// NETWORK 2
//   _strobeTimer.ET: elapsed time
Control.SystemTime.FastFlash := F_LIMIT(En := TRUE, High := 500, Value := TIME_TO_REAL(_strobeTimer.ET), Low := 0) OR F_LIMIT(En := TRUE, High := 1500, Value := TIME_TO_REAL(_strobeTimer.ET), Low := 1000);

// NETWORK 3
//   _strobeTimer.ET: elapsed time
Control.SystemTime.PulseFlash := F_LIMIT(En := TRUE, High := 1500, Value := TIME_TO_REAL(_strobeTimer.ET), Low := 1250) OR F_LIMIT(En := TRUE, High := 2000, Value := TIME_TO_REAL(_strobeTimer.ET), Low := 1750);

// NETWORK 4
//   _strobeTimer.ET: elapsed time
Control.SystemTime.SlowFlash := F_LIMIT(En := TRUE, High := 1000, Value := TIME_TO_REAL(_strobeTimer.ET), Low := 0);
END_ACTION

ACTION A_SyncSystemTime:
_fb_LocalSystemTime(sNetID := '', bEnable := TRUE, dwCycle := 15, dwOpt := 1, tTimeout := DEFAULT_ADS_TIMEOUT);
IF _fb_LocalSystemTime.bValid THEN
	Control.SystemTime.CurrentTime := _fb_LocalSystemTime.systemTime;
END_IF
END_ACTION

ACTION A_TimePulses:
//Second Pulse
_timer_ET := _timer_ET + DWORD_TO_DINT(_lastScanTime);
IF _timer_ET >= _ticksInSecond THEN 
	Control.SystemTime.SecondPulse := TRUE;
	Control.SystemTime.SecondsNow := TO_DWORD(SYSTEMTIME_TO_DT(Control.SystemTime.CurrentTime));
	_timer_ET := 0;
ELSE
	Control.SystemTime.SecondPulse := FALSE;
END_IF

//Minute Pulse
_MinutePulse(CLK := Control.SystemTime.CurrentTime.wSecond = 0);
Control.SystemTime.MinutePulse :=  _MinutePulse.Q;

//Hour Pulse
_HourPulse(CLK := Control.SystemTime.CurrentTime.wMinute = 0);
Control.SystemTime.HourPulse :=  _HourPulse.Q;

//Midnight Pulse
IF WORD_TO_INT(Control.SystemTime.CurrentTime.wDay) <> Control_SP.TimeManagement.PreviousDay THEN
	Control.SystemTime.MidnightPulse := TRUE;
	Control_SP.TimeManagement.PreviousDay := WORD_TO_INT(Control.SystemTime.CurrentTime.wDay);
ELSE
	Control.SystemTime.MidnightPulse := FALSE;
END_IF
END_ACTION

ACTION A_UpTime:
IF Control.SystemTime.SecondPulse THEN
	//Up time since last reset
	Control.SystemTime.UpTime.Seconds := Control.SystemTime.UpTime.Seconds + 1;
	IF Control.SystemTime.UpTime.Seconds >= 60 THEN 
		Control.SystemTime.UpTime.Minutes := Control.SystemTime.UpTime.Minutes + 1;
		Control.SystemTime.UpTime.Seconds := 0;
	END_IF
	IF Control.SystemTime.UpTime.Minutes >= 60 THEN 
		Control.SystemTime.UpTime.Hours := Control.SystemTime.UpTime.Hours + 1;
		Control.SystemTime.UpTime.Minutes := 0;
	END_IF
	IF Control.SystemTime.UpTime.Hours >= 24 THEN 
		Control.SystemTime.UpTime.Days := Control.SystemTime.UpTime.Days + 1;
		Control.SystemTime.UpTime.Hours := 0;
	END_IF
	
	//Total up time
	Control_SP.TimeManagement.TotalUpTime.Seconds := Control_SP.TimeManagement.TotalUpTime.Seconds + 1;
	IF Control_SP.TimeManagement.TotalUpTime.Seconds >= 60 THEN 
		Control_SP.TimeManagement.TotalUpTime.Minutes := Control_SP.TimeManagement.TotalUpTime.Minutes + 1;
		Control_SP.TimeManagement.TotalUpTime.Seconds := 0;
	END_IF
	IF Control_SP.TimeManagement.TotalUpTime.Minutes >= 60 THEN 
		Control_SP.TimeManagement.TotalUpTime.Hours := Control_SP.TimeManagement.TotalUpTime.Hours + 1;
		Control_SP.TimeManagement.TotalUpTime.Minutes := 0;
	END_IF
	IF Control_SP.TimeManagement.TotalUpTime.Hours >= 24 THEN 
		Control_SP.TimeManagement.TotalUpTime.Days := Control_SP.TimeManagement.TotalUpTime.Days + 1;
		Control_SP.TimeManagement.TotalUpTime.Hours := 0;
	END_IF
END_IF
END_ACTION

END_FUNCTION_BLOCK

// Objects/FB_TwinSAFE_V4_01/FB_TwinSAFE
FUNCTION_BLOCK FINAL FB_TwinSAFE EXTENDS FB_EventLogger
VAR_IN_OUT
	Control								: ST_System;
END_VAR
VAR
	_ComErr					AT %I*		: BOOL;
	_FbErr					AT %I*		: BOOL;
	_OutErr					AT %I*		: BOOL;
	_ComStartUp				AT %I*		: BOOL;
	_OtherErr				AT %I*		: BOOL;
	_State					AT %I*		: UINT;
	_Daig					AT %I*		: UINT;
	_FSOUTModule1Fault 		AT %I* 		: BOOL;
	_FSOUTModule2Fault 		AT %I* 		: BOOL;
	_FSOUTModule3Fault 		AT %I* 		: BOOL;
	_FSOUTModule4Fault 		AT %I* 		: BOOL;
	_FSOUTModule5Fault 		AT %I* 		: BOOL;
	_FSOUTModule6Fault 		AT %I* 		: BOOL;
	_FSOUTRelaisModuleFault AT %I*      : BOOL;
	_FSINModule1Fault		AT %I* 		: BOOL;
	_FSINModule2Fault		AT %I* 		: BOOL;
	_FSINModule3Fault		AT %I* 		: BOOL;
	_FSINModule4Fault		AT %I* 		: BOOL;
	_FSINModule5Fault		AT %I* 		: BOOL;
	_FSINModule6Fault		AT %I* 		: BOOL;
	_FSINModule7Fault		AT %I* 		: BOOL;
	_FSINModule8Fault		AT %I* 		: BOOL;
	_FSINModule9Fault		AT %I* 		: BOOL;
	_FSINModule10Fault		AT %I* 		: BOOL;
	_SafetyChainFault 	    AT %I*  	: BOOL;
	_SafetyInRun			AT %I*  	: BOOL;
	_Module1Fault			AT %I*  	: BOOL;
	_RunStop				AT %Q*		: BOOL;
	_ErrAck					AT %Q*		: BOOL;
	_SafetyInRunReturn		AT %Q*  	: BOOL;
	_ModuleFault					  	: BOOL;
	_Alarm								: BOOL;					
	_Warning							: BOOL;					
	_AlarmMute							: BOOL;					
	_AlarmNum							: DINT;					
	_WarningNum							: DINT;					
	_FaultTimer_ET						: REAL;	
	_r_Trig								: ARRAY[0..9] OF R_TRIG;
END_VAR
VAR PERSISTENT
	_Name								: STRING[15];				//Name for HMI
	_Description						: STRING[40];				//Description for HMI
	_FaultTimer_PT						: REAL;						//Fault timer preset time
END_VAR

M_Control();
M_AlarmMonitor();
M_WarningMonitor();

//Alarm mute reset
IF Control.Inputs.AlarmMuteReset THEN _AlarmMute := FALSE; END_IF

{attribute 'monitoring' := 'variable'}
PROPERTY PUBLIC Alarm : Bool
GET
Alarm := _Alarm;
END_GET
END_PROPERTY

{attribute 'monitoring' := 'variable'}
PROPERTY PUBLIC Description : String[40]
GET
Description := _Description;
END_GET
SET
_Description := Description;
END_SET
END_PROPERTY

{attribute 'monitoring' := 'variable'}
PROPERTY PUBLIC FaultTimer_ET : real
GET
FaultTimer_ET := _FaultTimer_ET;
END_GET
END_PROPERTY

{attribute 'monitoring' := 'variable'}
PROPERTY PUBLIC FaultTimer_PT : real
GET
FaultTimer_PT := _FaultTimer_PT;
END_GET
SET
_FaultTimer_PT := FaultTimer_PT;
END_SET
END_PROPERTY

METHOD PRIVATE M_AlarmMonitor
VAR_INPUT
END_VAR
VAR_INST
END_VAR
VAR_INST // added by the converter: edge detectors and wires of the graphical bodies
    _w1, _w2, _w3 : BOOL;
END_VAR
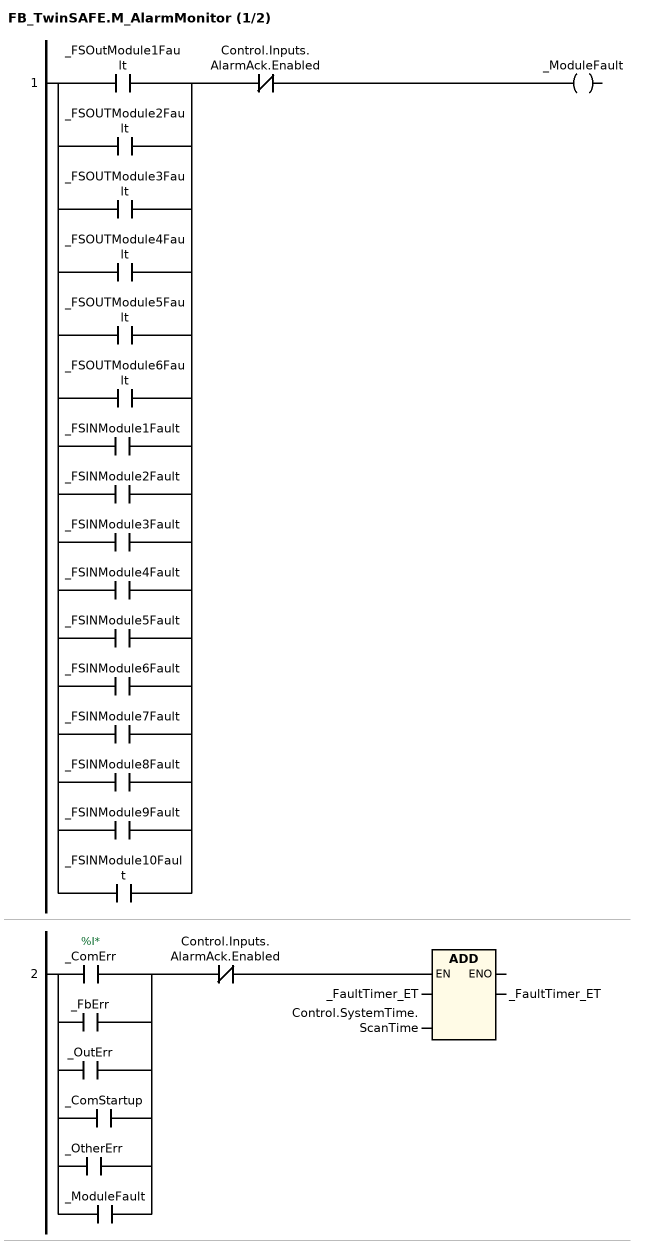
// NETWORK 1
_ModuleFault := (_FSOutModule1Fault OR _FSOUTModule2Fault OR _FSOUTModule3Fault OR _FSOUTModule4Fault OR _FSOUTModule5Fault OR _FSOUTModule6Fault OR _FSINModule1Fault OR _FSINModule2Fault OR _FSINModule3Fault OR _FSINModule4Fault OR _FSINModule5Fault OR _FSINModule6Fault OR _FSINModule7Fault OR _FSINModule8Fault OR _FSINModule9Fault OR _FSINModule10Fault) AND NOT Control.Inputs.AlarmAck.Enabled;

// NETWORK 2
//   _ComErr: AT %I*
//   _FaultTimer_ET: Fault timer elapsed
//   Control.SystemTime.ScanTime: Last scan time (Seconds)
IF (_ComErr OR _FbErr OR _OutErr OR _ComStartup OR _OtherErr OR _ModuleFault) AND NOT Control.Inputs.AlarmAck.Enabled THEN
    _FaultTimer_ET := _FaultTimer_ET + Control.SystemTime.ScanTime;
END_IF

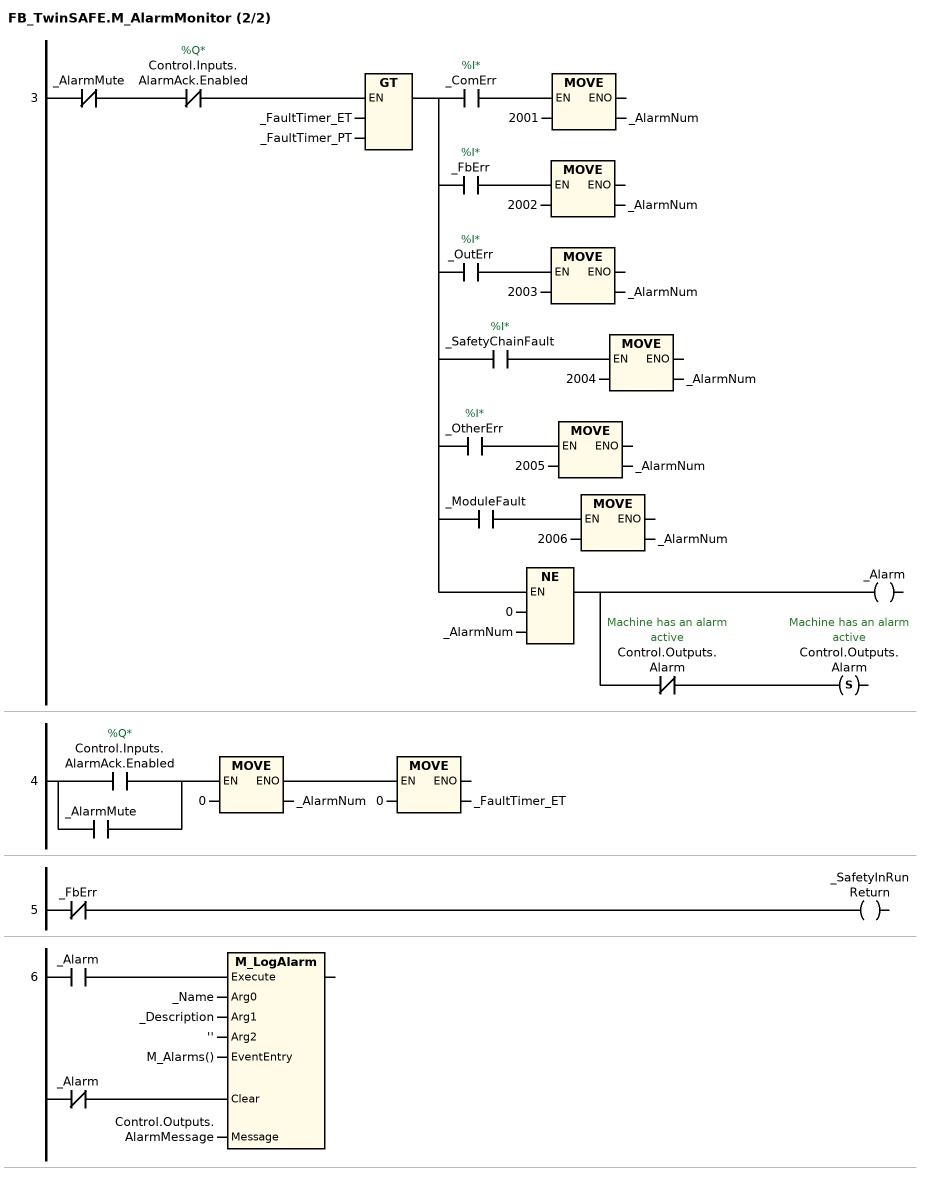
// NETWORK 3
//   Control.Inputs.AlarmAck.Enabled: AT %Q*
//   _ComErr: AT %I*
//   _FbErr: AT %I*
//   _OutErr: AT %I*
//   _SafetyChainFault: AT %I*
//   _OtherErr: AT %I*
//   Control.Outputs.Alarm: Machine has an alarm active
_w1 := NOT _AlarmMute AND NOT Control.Inputs.AlarmAck.Enabled AND _FaultTimer_ET > _FaultTimer_PT;
IF _w1 AND _ComErr THEN _AlarmNum := 2001; END_IF
IF _w1 AND _FbErr THEN _AlarmNum := 2002; END_IF
IF _w1 AND _OutErr THEN _AlarmNum := 2003; END_IF
IF _w1 AND _SafetyChainFault THEN _AlarmNum := 2004; END_IF
IF _w1 AND _OtherErr THEN _AlarmNum := 2005; END_IF
IF _w1 AND _ModuleFault THEN _AlarmNum := 2006; END_IF
_w2 := _w1 AND 0 <> _AlarmNum;
_Alarm := _w2;
Control.Outputs.Alarm S= _w2 AND NOT Control.Outputs.Alarm;

// NETWORK 4
//   Control.Inputs.AlarmAck.Enabled: AT %Q*
_w3 := Control.Inputs.AlarmAck.Enabled OR _AlarmMute;
IF _w3 THEN _AlarmNum := 0; END_IF
IF _w3 THEN _FaultTimer_ET := 0; END_IF

// NETWORK 5
_SafetyInRunReturn := NOT _FbErr;

// NETWORK 6
M_LogAlarm(Execute := _Alarm, Arg0 := _Name, Arg1 := _Description, Arg2 := '', EventEntry := M_Alarms(), Clear := NOT _Alarm, Message := Control.Outputs.AlarmMessage);
END_METHOD

METHOD PRIVATE M_Alarms : TcEventEntry
VAR_INPUT
END_VAR
VAR_INST
END_VAR
CASE _AlarmNum OF		
2001:	M_Alarms := 	TC_Events.TcTwinSafe.A_2001;//Communication Error			
2002:	M_Alarms := 	TC_Events.TcTwinSafe.A_2002;//Feedback Error			
2003:	M_Alarms := 	TC_Events.TcTwinSafe.A_2003;//Output Error	
2004:	M_Alarms := 	TC_Events.TcTwinSafe.A_2004;//Safety Chain Fault	    
2005:	M_Alarms := 	TC_Events.TcTwinSafe.A_2005;//Other Error	 
2006:	M_Alarms := 	TC_Events.TcTwinSafe.A_2006;//Module Error	                    	
ELSE                        	
		M_Alarms := 	TC_Events.TcTwinSafe.A_Undefined;
END_CASE
END_METHOD

METHOD PRIVATE M_Control
VAR_INPUT
END_VAR
VAR_INST
	_resetStep				: INT;
END_VAR
VAR_INST // added by the converter: edge detectors and wires of the graphical bodies
    _rt1 : R_TRIG;
    _w1 : BOOL;
END_VAR
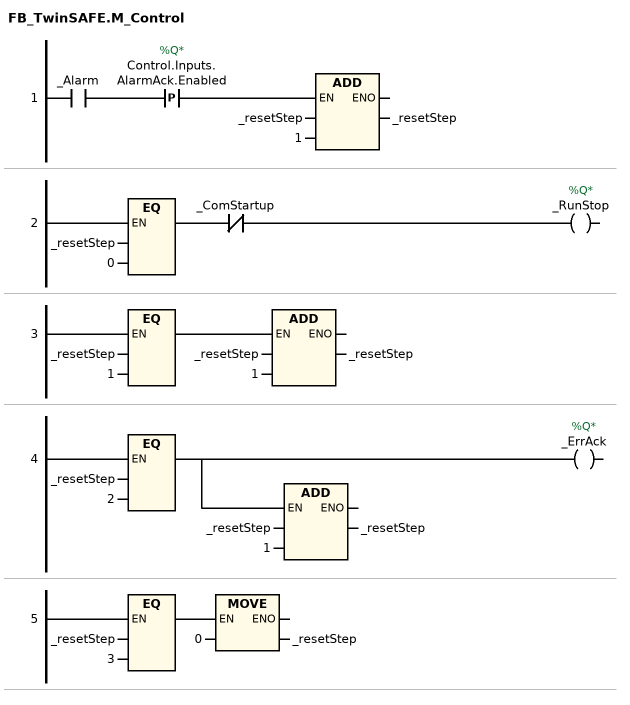
// NETWORK 1
//   Control.Inputs.AlarmAck.Enabled: AT %Q*
_rt1(CLK := Control.Inputs.AlarmAck.Enabled);
IF _Alarm AND _rt1.Q THEN _resetStep := _resetStep + 1; END_IF

// NETWORK 2
//   _RunStop: AT %Q*
_RunStop := _resetStep = 0 AND NOT _ComStartup;

// NETWORK 3
IF _resetStep = 1 THEN _resetStep := _resetStep + 1; END_IF

// NETWORK 4
//   _ErrAck: AT %Q*
_w1 := _resetStep = 2;
_ErrAck := _w1;
IF _w1 THEN _resetStep := _resetStep + 1; END_IF

// NETWORK 5
IF _resetStep = 3 THEN _resetStep := 0; END_IF
END_METHOD

METHOD PRIVATE M_WarningMonitor
VAR_INPUT
END_VAR
VAR_INST
END_VAR
VAR_INST // added by the converter: edge detectors and wires of the graphical bodies
    _w1, _w2 : BOOL;
END_VAR
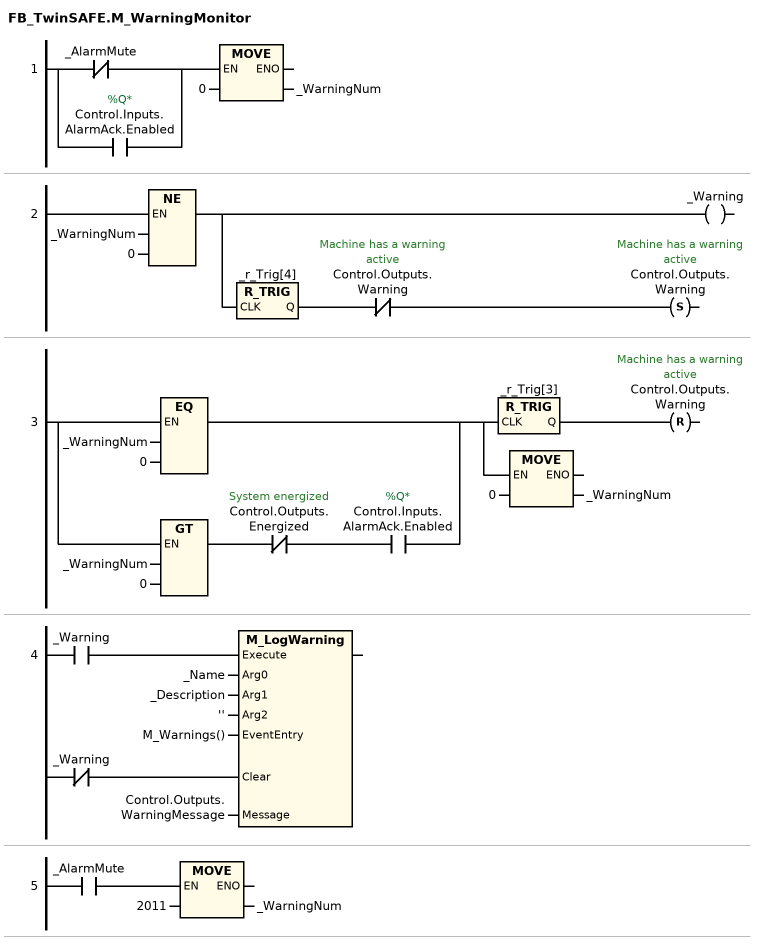
// NETWORK 1
//   Control.Inputs.AlarmAck.Enabled: AT %Q*
IF NOT _AlarmMute OR Control.Inputs.AlarmAck.Enabled THEN _WarningNum := 0; END_IF

// NETWORK 2
//   Control.Outputs.Warning: Machine has a warning active
_w1 := _WarningNum <> 0;
_Warning := _w1;
_r_Trig[4](CLK := _w1); // R_TRIG
Control.Outputs.Warning S= _r_Trig[4].Q AND NOT Control.Outputs.Warning;

// NETWORK 3
//   Control.Outputs.Energized: System energized
//   Control.Inputs.AlarmAck.Enabled: AT %Q*
//   Control.Outputs.Warning: Machine has a warning active
_w2 := _WarningNum = 0 OR _WarningNum > 0 AND NOT Control.Outputs.Energized AND Control.Inputs.AlarmAck.Enabled;
_r_Trig[3](CLK := _w2); // R_TRIG
Control.Outputs.Warning R= _r_Trig[3].Q;
IF _w2 THEN _WarningNum := 0; END_IF

// NETWORK 4
M_LogWarning(Execute := _Warning, Arg0 := _Name, Arg1 := _Description, Arg2 := '', EventEntry := M_Warnings(), Clear := NOT _Warning, Message := Control.Outputs.WarningMessage);

// NETWORK 5
IF _AlarmMute THEN _WarningNum := 2011; END_IF
END_METHOD

METHOD PRIVATE M_Warnings : TcEventEntry
VAR_INPUT
END_VAR
VAR_INST
END_VAR
CASE _WarningNum OF
	2011:   M_Warnings :=	TC_Events.TcTwinSafe.W_2011;//Alarm Mute Active			
ELSE
	M_Warnings := 	TC_Events.TcTwinSafe.W_Undefined;
END_CASE
END_METHOD

{attribute 'monitoring' := 'variable'}
PROPERTY PUBLIC Name : String[15]
GET
Name := _Name;
END_GET
SET
_Name := Name;
END_SET
END_PROPERTY

{attribute 'monitoring' := 'variable'}
PROPERTY PUBLIC Warning : Bool
GET
Warning := _Warning;
END_GET
END_PROPERTY

END_FUNCTION_BLOCK
